ABB RAPID module: TG_Comms.sys

MODULE TG_Comms(SYSMODULE)
    !***********************************************************************
    ! TetraGen HMI request library for ABB - Phase 1 (comm core)
    !
    ! RAPID port of the FANUC KAREL request programs.
    ! Design & wire protocol: docs/abb_port_plan_v1.md
    !
    ! Loaded resident in task T_ROB1. The .tgs program modules (loaded
    ! dynamically by TG_Main in Phase 3) call the TG_* PROCs and read the
    ! shared PERS data below directly - RAPID's task-wide global scope makes
    ! every non-LOCAL symbol of a loaded module visible to all other modules.
    !
    ! Naming:  TG_*  = public API (called by TG_Main and .tgs programs)
    !          tg*   = internal helpers (LOCAL)
    !
    ! Wire protocol: byte-compatible with the FANUC TGS HMI protocol
    ! (request ids, prompts, 1-byte "0" acks, fixed-width scalars) EXCEPT
    ! frame/pose payloads, which travel as RAPID pose literals
    ! "[[x,y,z],[q1,q2,q3,q4]]" with a normalized quaternion (plan 4.5).
    !
    ! Tool/frame parameter style (plan 7.6, decided 2026-08-28): the pose-
    ! reporting request PROCs take explicit \Tool/\WObj PERS parameters
    ! (option b - the frame is visible at every call site, and a PERS
    ! parameter is itself a persistent reference, so it feeds CRobT
    ! directly). The FANUC-style modal numbers (nTG_ActTool/nTG_ActFrame)
    ! remain as a DEPRECATED fallback for calls that omit the arguments -
    ! kept deliberately as the back-pocket alternative; do not delete.
    !***********************************************************************

    ! ------------------------------------------------------------------
    ! Connection config. Edit from FlexPendant/RobotStudio, no code change.
    ! Virtual controller: keep "127.0.0.1". Real IRC5: the controller LAN IP.
    PERS string stTG_ServerIP:="127.0.0.1";
    PERS num nTG_Port:=2000;

    ! Settle time (s) applied after WaitRob and before every reported pose.
    ! VC measurements (findings doc): WaitRob \InPos alone left up to ~2 mm
    ! of residual convergence; 0.2 s reaches full settle (and matches the
    ! FANUC WAIT 0.20 before R_C). Tune from the data view without reloading
    ! code; on the real cell it also covers mechanical vibration damping.
    PERS num nTG_SettleTime:=0.2;

    ! ------------------------------------------------------------------
    ! Shared state: FANUC register-map equivalents (plan 4.3).
    PERS string stTG_ProgPass:="none";     ! SR[24] program name == project password
    PERS string stTG_SubName:="none";      ! SR[25] sub-routine token
    PERS string stTG_RobStatus:="Ok";      ! SR[23] robot status string
    PERS string stTG_ProgName:="none";     ! prog name received by TG_ReqFileTransfer
    PERS num nTG_ProgSel:=0;               ! R[188] 1=run .tgs program, 2=camera calibration
    PERS num nTG_FtpStatus:=0;             ! R[189] file transfer ok
    PERS num nTG_PassOK:=0;                ! R[200] password correct
    PERS num nTG_DryRun:=0;                ! R[199] dry-run flag
    PERS num nTG_DoCapture:=0;             ! R[197] do-capture flag; 2 = robot-side abort sentinel (matrix I4)
    PERS num nTG_CaptureOK:=0;             ! R[196] capture succeeded
    PERS num nTG_GlobalCapOK:=0;           ! R[187] global captures done status
    PERS num nTG_WeldStatus:=0;            ! R[198] 0=skip weld, 1=weld, 2=abort program
    PERS num nTG_UdwpFlag:=0;              ! R[170] user-defined weld params flag
    PERS num nTG_WelderType:=0;            ! 1=Miller, 2=FroniusTPSi (KAREL local var)
    PERS num nTG_WeldProc:=0;              ! R[171] weld procedure number
    PERS num nTG_WireFeed:=0;              ! R[172] wire feed speed
    PERS num nTG_ArcLength:=0;             ! R[173] arc length
    PERS num nTG_ArcControl:=0;            ! R[174] arc control
    PERS num nTG_TravelSpeed:=0;           ! R[175] travel speed

    ! ---- WS3/WS4 (2026-09-20): the values ABB needs and FANUC does not -----
    ! ABB takes weld parameters from the PROGRAM, not from a numbered schedule
    ! on the controller, so the HMI must serve the whole set on every weld -
    ! see the R_W_P note in TG_ReqWeldParams. Two additions carry what the
    ! FANUC wire never had to:
    !
    ! nTG_WeldSched is the POWER SOURCE's program / characteristic number,
    ! which lands in welddata main_arc.sched. It is NOT the FANUC "schedule
    ! number" of WELD START[proc,sched] (that selects a row in an ArcTool
    ! schedule file, a concept ABB has no equivalent of); it is the number the
    ! Fronius/Miller uses to pick a synergic line. MONARCH's own welddata
    ! records carry 1, 2 and 4 here.
    PERS num nTG_WeldSched:=0;             ! -> welddata main_arc.sched
    ! The seam phases: the parts of a weld either side of the steady arc.
    ! MONARCH's mDeclarations.sys carries ~15 distinct seamdata records that
    ! differ almost entirely in these, so a preset that cannot express them
    ! cannot reproduce their welds. Times in SECONDS, wire feeds in IPM and
    ! volts absolute - the same units the rest of this wire uses; TG_Weld.sys
    ! does the conversion, this module only stores.
    PERS num nTG_PurgeTime:=0;             ! -> seamdata purge_time
    PERS num nTG_PreflowTime:=0;           ! -> seamdata preflow_time
    PERS num nTG_PostflowTime:=0;          ! -> seamdata postflow_time
    PERS num nTG_BurnbackTime:=0;          ! -> seamdata bback_time
    PERS num nTG_CraterFillTime:=0;        ! -> seamdata fill_time
    PERS num nTG_CraterFillWireFeed:=0;    ! -> seamdata fill_arc.wirefeed
    PERS num nTG_CraterFillVolts:=0;       ! -> seamdata fill_arc.voltage
    PERS num nTG_IgnitionWireFeed:=0;      ! -> seamdata ign_arc.wirefeed
    PERS num nTG_IgnitionVolts:=0;         ! -> seamdata ign_arc.voltage

    ! Phase 7 (2026-09-04): pendant touch-up offset mirror (FANUC R[180..182],
    ! r_w_f.kl of the same date). The HMI pushes its stored per-weld touch-up
    ! offset on EVERY weld-frame reply - weld, skip and abort alike -
    ! so this always mirrors HMI state for the weld last served ("registers
    ! are a mirror, never a store", HMI docs/pendant_touchup_hmi_plan_v1.md).
    ! RECEIVE-AND-STORE ONLY: nothing on the ABB side consumes it yet - the
    ! FlexPendant entry/send path (FANUC R_O_T, id 20) is not ported.
    ! Units: INCHES verbatim off the wire (their D4), converted nowhere.
    PERS pos posTG_Touchup:=[0,0,0];       ! R[180..182] X/Y/Z, inches

    ! Phase 6: R_W_S weld statistics. No FANUC register equivalent - KAREL
    ! read the ArcTool record $AWEWELDSTAT[1] directly (R_W_S.kl). An IRC5
    ! has no drop-in equivalent of that record, so the .tgs program writes
    ! these three PERS just before calling TG_ReqWeldStats.
    ! TODO: DUMMY VALUES - the .tgs programs currently write fixed numbers to
    ! mimic the sensing. Producing REAL values is its own task; the candidate
    ! sources are listed in docs/abb_weld_stats_port_v1.md section 6. Only the
    ! source of the numbers changes then - the wire below is final.
    ! Units are fixed by the HMI, not by us: distance in mm (it divides by
    ! 25.4 for its analytics, which take inches) and time in seconds.
    PERS num nTG_WeldDist:=0;              ! $WELD_DIST   welded distance, mm
    PERS num nTG_ArcOnTime:=0;             ! $ARC_ON_TIME arc-on time, s
    ! 1 = the arc really ran. The HMI tests this for equality with 1, so it is
    ! a FLAG here, never a count - see the doc's 1.4 for why that distinction
    ! is not merely theoretical on the FANUC side.
    PERS num nTG_SuccArcEnd:=0;            ! $SUCC_AE

    ! Phase 5 (touch-up/retrieval doc section 4): 1 = an operator-edited
    ! .tgs module was detected at unload and staged in HOME:/TGS/edited/
    ! for the HMI's "Retrieve robot program from controller". No FANUC
    ! register equivalent (FANUC needs none: its MD: memory device serves
    ! the touched-up program directly). Set by tgSaveEditedModule
    ! (TG_Main); cleared by the HMI/tg_retrieve.py after a successful
    ! retrieval (RWS symbol write) - the robot never clears it.
    PERS num nTG_ProgEdited:=0;

    ! Frames received from the HMI (FANUC PR[5]/UFRAME[5], PR[6]/UFRAME[6]).
    ! Request PROCs write .oframe; the .tgs program references these wobjs in
    ! its move instructions - no separate "activate" step exists or is needed
    ! FOR THE TWO BASE-REFERENCED OBJECTS. The coordinated shape is another
    ! story: its station must be an ACTIVE mechanical unit (ActUnit) before
    ! a move - or a CRobT - in that work object resolves. That is one of the
    ! coordinated prerequisites still open; see the WIP block below.
    !
    ! THE RULE (weld_frame_update_strategy_v1, 2026-09-03).
    ! A request writes .oframe, ALWAYS - one write target, no case to
    ! detect here. What the HMI SENDS branches on one thing only: whether
    ! the weld is coordinated.
    !
    !   NOT COORDINATED - static table, OR indexed on a 1-/2-axis
    !   positioner that does not move during the weld:
    !       ufprog TRUE, ufmec "", uframe identity
    !       oframe <- the CAD/part frame W.R.T. THE ROBOT BASE
    !       (exactly what the HMI sends FANUC today)
    !
    !   COORDINATED MOTION - WORK IN PROGRESS, see the declaration below:
    !       ufprog FALSE, ufmec "<station>", uframe computed live by the
    !       controller from the station angles (the declared one ignored)
    !       oframe <- OPEN: the part W.R.T. THE POSITIONER FRAME, or a
    !       DISPLACEMENT in that frame, which is what the HMI's own
    !       (unfinished, untested) coordinated FANUC path computes today
    !
    ! Writing THE SERVED FRAME to uframe is never right. Coordinated: the
    ! controller ignores uframe outright (plan E28), so the write is a
    ! SILENT no-op - finding F-2's failure mode. Not coordinated: uframe is
    ! identity, so writing oframe is the same geometry anyway, because
    ! motion and CRobT both see only the product uframe*oframe.
    !
    ! BUT "uframe is identity" is a claim about the LIVE PERS VALUE, not
    ! about the declarations below. A PERS keeps whatever it was last
    ! assigned - across program loads, and across a saved station - so a
    ! controller that ever ran the pre-2026-09-03 code, which served the
    ! frame INTO uframe, still holds that frame there. Compose it with the
    ! new oframe write and every pose is double-transformed silently, while
    ! a pendant watch on oframe shows exactly the expected numbers.
    ! => AN EXPORTED PROGRAM MUST ASSIGN uframe:=IDENTITY AT ENTRY, next to
    ! its .oframe nominal, for every base-referenced work object it uses.
    ! That is a one-time normalization of an assumption, NOT a frame write,
    ! and it is the one legitimate reason to touch uframe at all.
    ! TD05Test.mod and TD05Weld.mod both do it; THE WELD PLANNER ABB
    ! EXPORTER MUST TOO.
    !
    ! ONE DECLARATION PER SHAPE - ufprog/ufmec ARE NEVER WRITTEN AT RUNTIME.
    ! The two shapes are separate symbols, so a program picks one by PASSING
    ! it (\WObj:=...) rather than by mutating a record. Reasons, in order:
    !   - runtime ufmec re-binding is unverified and unusual; declaring each
    !     shape once makes the question moot;
    !   - a program mixing indexed and coordinated welds would otherwise
    !     have to reassign mid-run, which is exactly the look-ahead hazard
    !     tracked as O-3 (a PERS write landing after RAPID has already
    !     prepared queued instructions);
    !   - robtargets bind by NAME, so a record whose kind changes mid-program
    !     makes the same named target mean different things at different
    !     points - and a pendant watch shows one mutating record;
    !   - the static shape stays byte-identical to what a VC has accepted.
    ! An exported program therefore assigns only frame COMPONENTS at entry -
    ! .uframe identity and .oframe nominal - never ufprog/ufmec.
    ! EXCEPTION (2026-09-23, VC-proven): wobjTG_WeldActStn below is bound
    ! at run time by TG_ActMechUnit - once, at module entry, before any
    ! motion - so one coordinated program can run on either station. It is a
    ! separate record, always coordinated, so none of the reasons above bite.
    ! NOTE Accepted cost: ufprog/ufmec correctness
    ! now lives on the controller, the same trust model as tTG_Weld - a
    ! wrong ufmec here is a silent wrong-station weld, so treat these as
    ! cell configuration and verify them when commissioning.
    !
    ! For an INDEXED weld the served frame describes the part AT THE ANGLE
    ! THE WELD PLANNER AUTHORED for that weld: the HMI rotates its
    ! localization result from the capture angle to the weld's
    ! tool_path_parameters positioner_angle - bTpos * Rz(dtheta) *
    ! inverse(bTpos) - and NEVER reads the robot's actual station position.
    ! So the served value does not depend on when the request runs, and the
    ! real requirement is that THE PROGRAM'S INDEX EQUALS THE ANGLE THE
    ! PLANNER AUTHORED (true by construction for an exported program).
    ! Keep the safe order regardless: index, then request the frame, then
    ! weld. And once a frame has been served, do not re-assign either
    ! component before the weld that consumes it.
    !
    ! ---- Non-coordinated: static table, or indexed on a positioner -------
    ! Base-referenced. Identity uframe, so uframe*oframe = oframe = whatever
    ! the HMI serves. These are also the standalone/VC defaults.
    PERS wobjdata wobjTG_Cam:=[FALSE,TRUE,"",[[0,0,0],[1,0,0,0]],[[0,0,0],[1,0,0,0]]];
    PERS wobjdata wobjTG_Weld:=[FALSE,TRUE,"",[[0,0,0],[1,0,0,0]],[[0,0,0],[1,0,0,0]]];

    ! ---- Coordinated motion, one work object per station -----------------
    ! WORK IN PROGRESS on both sides of the wire, 2026-09-03. These are the
    ! declared shapes only; nothing in this repo references them yet, and the
    ! prerequisites listed at the end of this block are all still open.
    ! UPDATE 2026-09-12: the oframe CONVENTION is no longer open - it is
    ! ABSOLUTE, see below - and the PC-side exporter now passes these records
    ! by name (curobo_suite D47). The prerequisites below are unchanged and
    ! still open, and nothing here has been loaded on a controller.
    !
    ! ufprog FALSE + ufmec => the controller derives uframe live from the
    ! station angles and IGNORES the declared uframe, which is why it is
    ! left identity. oframe is the component TG_ReqWeldFrame writes.
    !
    ! COMMENT THESE DECLARATIONS OUT WHEN THE TEST CELL HAS NO EXTERNAL AXIS,
    ! or change "STN1"/"STN2" to the mechanical units of the setup being
    ! tested - and comment out the second one on a single-station cell.
    ! Each name must exist in this controller's MOC configuration, and the
    ! phase 1-6 validation VC (RW6.15.08/IRB4600) has no positioner at all.
    ! THIS FILE IS THE SHARED SYSMODULE: if a controller rejects an
    ! unresolvable ufmec at load or at Check Program, it takes the ALREADY
    ! VALIDATED non-coordinated path down with it - and there are now TWO
    ! names that can do that. One "!" in front of each declaration line is
    ! the whole rollback. Note the asymmetry - an unresolvable name fails
    ! loudly, while a wrong-but-resolvable one is a silent wrong-station
    ! weld, so verify BOTH names at commissioning. Two declared stations
    ! make that silent case reachable on a correctly built cell for the
    ! first time: STN1/STN2 transposed welds the right geometry on the
    ! wrong table, where with one station declared a mix-up could only ever
    ! fail loudly.
    ! NOTE NOT YET LOADED ON A CONTROLLER. Only the static shape above has been
    ! (LOCAL PERS wobjdata accepted as a \WObj argument, RW6.15.08/IRB4600,
    ! Check Program clean). Bundle this with the coordinated VC load-check.
    !
    ! WHAT THIS oframe CARRIES - RESOLVED 2026-09-12 as ABSOLUTE: the
    ! CORRECTED PART POSE IN THE WORK OBJECT'S USER FRAME, which for these
    ! records is the station. Not a displacement. Decision is curobo_suite
    ! plan D47; full reasoning and the rejected alternative are in
    ! curobo_suite docs/abb_coordinated_hmi_frame_contract_v1.md.
    !
    ! The deciding argument is SLOT COUNT, not geometry. FANUC can afford a
    ! displacement because it has TWO runtime registers - the absolute goes
    ! to the UFRAME PR and the delta to the OFFSET PR, two slots with two
    ! meanings that cannot collide. Here there is ONE writable frame, and
    ! .oframe is ALSO where the non-coordinated absolute lands, because
    ! TG_ReqWeldFrame writes it unconditionally on whatever it is handed
    ! (the O-1 resolution). Under a displacement convention that one slot
    ! would mean "absolute" for wobjTG_Weld and "delta" for
    ! wobjTG_WeldStn<n>, with NO ERROR when the two are swapped. Absolute
    ! gives one sentence covering both records and keeps RAPID free of case
    ! detection. ABB's own MultiMove manual reads the same way: its
    ! wobj_stn1 example puts the part's mounting offset in oframe.
    !
    ! A displacement is NOT geometrically impossible - it works if the
    ! exporter re-encodes the robtargets into the positioner flange frame,
    ! which is exactly what the FANUC path does. So this was a cost and
    ! coupling decision, not a correctness one, and section 7 of
    ! docs/abb_coordinated_weld_hmi_plan_v1.md (curobo_suite) records what
    ! would reopen it: a decision to keep getWeldFrameToSendToRobot
    ! brand-blind.
    !
    ! WHAT THE HMI STILL HAS TO DO. RobotCell::getWeldFrameToSendToRobot is
    ! brand-agnostic today and returns
    ! Weld::GetCoordinatedOffsetInPositionerFrame - the FANUC DISPLACEMENT -
    ! for every coordinated weld. Fed to TG_ReqWeldFrame that produces a
    ! module which loads, runs, and welds in the wrong place with no error.
    ! That call site must branch on brand IN THE SAME CHANGE that enables
    ! coordinated ABB welds. The correct value is the existing offset
    ! composed onto the nominal: offset_in_pos * (inv(P) * C_nom) =
    ! inv(P) * C_cor, exact, and C_nom cancels.
    !
    ! Prerequisites, none of them closed (all WIP):
    !   - ActUnit for the station, and whether it is a mechanical unit in
    !     the robot's own motion task or a MultiMove group (SyncMoveOn);
    !   - real extjoint values for the station axes in every robtarget -
    !     the exporter writes 9E9 for axes it does not command (plan D5);
    !   - the controller's STN1 and STN2 BASE FRAMES must EACH agree with
    !     the positioner calibration the PC uses. A disagreement is a silent
    !     rigid offset on every coordinated weld on THAT station - E47 one
    !     level up, and a bigger risk than a mistyped ufmec. Two stations is
    !     two independent calibrations to verify, not one checked twice.
    PERS wobjdata wobjTG_WeldStn1:=[FALSE,FALSE,"STN1",[[0,0,0],[1,0,0,0]],[[0,0,0],[1,0,0,0]]];
    ! Station 2 (D4's two-station template). Same shape, different ufmec, and
    ! a SEPARATE resident symbol for exactly the reason Stn1 is separate from
    ! wobjTG_Weld: ufmec is baked into the record and is never re-bound at
    ! runtime, so one work object cannot serve both stations. Each station is
    ! declared once here and an exported program picks one BY PASSING IT -
    ! TG_ReqWeldFrame writes .oframe on whatever it is handed - so which
    ! station a weld belongs to is expressed entirely at the call site:
    !     TG_ReqWeldFrame \Tool:=tTG_Weld \WObj:=wobjTG_WeldStn2;
    ! The two oframes are independent slots and serving one never touches the
    ! other, so a program alternating stations does not disturb a frame it
    ! already holds for the other one. Everything above applies unchanged:
    ! same oframe convention (ABSOLUTE, resolved 2026-09-12), same
    ! prerequisites, same rollback.
    !
    ! TWO PREREQUISITES THAT ONLY EXIST ONCE THERE ARE TWO STATIONS, both
    ! read off the MONARC teardown of a real IRBP D600 two-station cell
    ! (customer_specific/monarc/, joint_limits.md and monarc_cell_teardown.html):
    !   - THE STATIONS CANNOT BOTH BE ACTIVE. Five positioner motors share
    !     three drives through contactors K1-K5, so ActUnit STN2 requires
    !     DeactUnit STN1 first. Declaring both work objects is fine -
    !     declaring is not activating - but only the ACTIVE station's object
    !     resolves for a move or a CRobT. A two-station program brackets
    !     each station's work in ActUnit/DeactUnit.
    !   - THE extjoint SLOTS ARE SHARED. eax_b/eax_c are ARM1/PLATE1 or
    !     ARM2/PLATE2 depending on which unit is active, because the logical
    !     axis numbers are reused. A robtarget carried from a station-1
    !     program into a station-2 one commands station 2's axes to station
    !     1's angles WITHOUT COMPLAINT. That lands on the exporter (plan
    !     D5), not here, but it is the same silent-wrong-station family as
    !     a transposed ufmec.
    ! NOTE "STN1"/"STN2" are the actual configured unit names in that cell,
    ! which is the best evidence available that these are the right strings -
    ! but neither has been checked against the target controller's MOC, so
    ! treat both as unverified until commissioning.
    ! NOTE The MONARC feasibility note proposes moving the coordinated objects
    ! out into a per-cell TG_Frames.sys adapter, on the grounds that station
    ! names are cell configuration rather than generic core. That split has
    ! not been taken; if it is, both declarations move together.
    PERS wobjdata wobjTG_WeldStn2:=[FALSE,FALSE,"STN2",[[0,0,0],[1,0,0,0]],[[0,0,0],[1,0,0,0]]];

    ! ---- Coordinated motion, "the station at the robot" -------------------
    ! 2026-09-23, VC-proven: ONE coordinated work object for
    ! whichever station is presented, so a coordinated program names no
    ! station and can run on both. Declared UNBOUND (ufmec ""): TG_ActMechUnit
    ! (TG_Cell.sys) writes ufmec from the SAME decision that activates the
    ! unit, on every call, before the program's first motion. Measured on the
    ! ProjectMonarch VC (RW 6.15, socket plan V-36):
    !   - ufmec "" loads; used unbound, CRobT stops the program (41450);
    !   - bound to the active station, a coordinated MoveL follows it: the
    !     station frame turned exactly with the chuck (9.961 deg for 9.961);
    !   - bound to the INACTIVE station, CRobT only LOGS 50066 and returns a
    !     pose that is not station-relative - execution continues - and the
    !     next coordinated move stops with 50066. No wrong-station motion;
    !   - a unit name the controller does not have stops the program (41450).
    ! The per-station records above stay for programs that name a station.
    PERS wobjdata wobjTG_WeldActStn:=[FALSE,FALSE,"",[[0,0,0],[1,0,0,0]],[[0,0,0],[1,0,0,0]]];

    ! No coordinated CAMERA work object, deliberately. Captures stay
    ! base-referenced on ABB exactly as on FANUC, so the HMI's scan and
    ! registration path is one code path across both brands (owner call,
    ! 2026-09-03). What that costs is a known, accepted accuracy item, not an
    ! oversight. See weld_frame_update_strategy_v1.md section 5, and for the
    ! two ways in if measurement later says it matters.
    !
    ! CORRECTION 2026-09-12 - the conditioning argument this note used to
    ! make does not survive measurement, and the convention it hedged on is
    ! now settled (see the coordinated block above). It read:
    !
    !   "What that costs depends on the open convention question above.
    !    Under the ABSOLUTE reading the PC's positioner model enters as a
    !    single left-multiply - inverse(plate_pc(theta_s)) * P_base - so a
    !    calibration error there lands on the weld at full magnitude. Under
    !    the DISPLACEMENT reading it enters as a conjugation that cancels at
    !    zero correction, which is the better-conditioned arithmetic."
    !
    ! Tested rather than argued. Model the station miscalibration as
    ! plate_ctrl(theta) = Y * plate_pc(theta) with Y = 3 mm + 0.2 deg, over a
    ! 7-sample 2-axis sweep with the tilt parked at 37 deg. Both conventions
    ! are wrong by EXACTLY THE SAME AMOUNT - 7.047 mm with no correction,
    ! 7.056 mm with a 2.6 mm correction - and both are exact (1e-12 mm) on a
    ! calibrated station. They are algebraically identical under that error
    ! mode, because Y left-multiplies the whole chain either way:
    ! plate_ctrl(theta) * oframe * p == plate_ctrl(theta) * delta * q for the
    ! corresponding point encodings.
    !
    ! The conjugation DOES cancel at zero correction - but what it cancels is
    ! the CORRECTION term, and the dominant term is the part's nominal
    ! placement, which crosses the PC/controller frame boundary exactly once
    ! in both conventions. So displacement buys no robustness here, and the
    ! absolute convention costs none.
    !
    ! WHAT THIS DOES NOT COVER, and is still open: an error in how the PC
    ! models the plate's MOTION - axis direction or offset, i.e. a
    ! theta-DEPENDENT mismatch rather than a constant Y. That was not tested
    ! and is a different question. If that is the real concern, measure it
    ! the same way before acting on it; the constant-Y result says nothing
    ! about it either way.

    ! Tools (FANUC UT[2] camera / UT[8] torch).
    ! TODO: DUMMY VALUES - replace with the calibrated tooldata of the real cell.
    PERS tooldata tTG_Cam:=[TRUE,[[0,0,100],[1,0,0,0]],[1,[0,0,50],[1,0,0,0],0,0,0]];
    PERS tooldata tTG_Weld:=[TRUE,[[0,0,200],[1,0,0,0]],[1,[0,0,100],[1,0,0,0],0,0,0]];

    ! DEPRECATED (plan 7.6, decided 2026-08-28) - FANUC modal
    ! UTOOL_NUM/UFRAME_NUM emulation: the .tgs program selects the active
    ! tool/frame BY NUMBER; tgSendPose resolves the number to the LIVE
    ! tooldata/wobjdata at read time. Superseded by explicit \Tool/\WObj
    ! PERS parameters on the request PROCs (style b), which make the frame
    ! visible at the call site instead of hidden global state. Only used
    ! when a request is called WITHOUT the arguments. Kept deliberately as
    ! the back-pocket alternative; do not delete.
    ! (A PERS-to-PERS copy would go stale when a request updates the frame -
    ! the same hazard FANUC handles by re-emitting UFRAME[n]=PR[n] after
    ! every frame-PR-writing routine. Numbers need no refresh.)
    PERS num nTG_ActTool:=8;               ! UTOOL_NUM:  2=camera, 8=torch
    PERS num nTG_ActFrame:=0;              ! UFRAME_NUM: 5=camera, 6=weld, else base

    ! Scratch persistents for CRobT: its \Tool/\WObj are PERS parameters
    ! (a VAR or FUNC result is rejected with Argument error 123). Only the
    ! DEPRECATED modal fallback needs them (tgActTool/tgActWobj are FUNCs,
    ! their results are values); the explicit style passes the caller's
    ! PERS parameters straight to CRobT, no scratch copy involved.
    ! tgSendPose refreshes them from the live data on every fallback call,
    ! so they cannot go stale. Internal - never reference in .tgs programs.
    LOCAL PERS tooldata tTG_Scratch:=[TRUE,[[0,0,200],[1,0,0,0]],[1,[0,0,100],[1,0,0,0],0,0,0]];
    LOCAL PERS wobjdata wobjTG_Scratch:=[FALSE,TRUE,"",[[0,0,0],[1,0,0,0]],[[0,0,0],[1,0,0,0]]];

    ! ------------------------------------------------------------------
    ! Socket state. Lifecycle owned by TG_Main via TG_SocketCom/TG_SocketDisc;
    ! .tgs programs must never touch these directly.
    LOCAL VAR socketdev tg_server_socket;
    LOCAL VAR socketdev tg_client_socket;
    LOCAL VAR string tg_client_ip:="";


    !===================================================================
    ! Socket lifecycle (FANUC: SOCKET_COM / SOCKET_DISC)
    !===================================================================

    PROC TG_SocketCom()
        ! FANUC: SOCKET_COM - (re)start the server and wait for the HMI client.
        ! SocketClose is safe on sockets that were never opened (RoboDK driver
        ! uses the same close-before-create pattern on RW5/6).
        SocketClose tg_server_socket;
        SocketClose tg_client_socket;
        SocketCreate tg_server_socket;
        SocketBind tg_server_socket,stTG_ServerIP,nTG_Port;
        SocketListen tg_server_socket;
        TPWrite "TG: waiting for HMI on port "\Num:=nTG_Port;
        SocketAccept tg_server_socket,tg_client_socket\ClientAddress:=tg_client_ip,\Time:=WAIT_MAX;
        TPWrite "TG: HMI connected: "+tg_client_ip;
    ERROR
        ! Error matrix F-A/I1: RAPID's retry counter is bounded by the
        ! system parameter "No Of Retry" (default 4) - without
        ! ResetRetryCount a handful of consecutive failures would stop the
        ! whole server loop. Resetting makes this reconnect loop indefinite
        ! (same idiom as the RoboDK driver). Pacing comes from WaitTime /
        ! the blocking SocketAccept, so this cannot busy-loop.
        IF ERRNO=ERR_SOCK_TIMEOUT THEN
            ResetRetryCount;
            RETRY;
        ELSEIF ERRNO=ERR_SOCK_CLOSED THEN
            SocketClose tg_server_socket;
            SocketClose tg_client_socket;
            WaitTime 2;
            ResetRetryCount;
            RETRY;
        ENDIF
    ENDPROC

    PROC TG_SocketDisc()
        ! FANUC: SOCKET_DISC - drop the HMI connection (and the listener; it is
        ! re-created by the next TG_SocketCom). WaitTime lets the TCP stack
        ! release the port before rebinding (RoboDK COM_End pattern).
        SocketClose tg_server_socket;
        SocketClose tg_client_socket;
        WaitTime 2;
        TPWrite "TG: socket disconnected";
    ENDPROC


    !===================================================================
    ! Wire-protocol helpers (plan 4.4)
    !===================================================================

    LOCAL PROC tgCycleAbort()
        ! FIX 2026-08-28 (error-recovery matrix F-F): bottom-level recovery
        ! for wire errors. VC evidence (kill test, RW 6.15): an unhandled
        ! error does NOT propagate through the late-binding call
        ! (%stTG_ProgName%) - the program STOPPED at the failing
        ! SocketReceive (events 41595/40228), so the tgRunTgsProgram /
        ! tgMainCycle handlers can never see a wire error raised inside a
        ! .tgs run. Recover where the error is born instead: log, drop the
        ! sockets, ExitCycle. PP moves to the start of main, which begins
        ! with TG_SocketDisc and loops back to accept - no propagation
        ! involved, works from any call depth (VC-validated 2026-08-28).
        ! VC-observed: ExitCycle's PP move does NOT drop \Dynamic modules
        ! (unlike a FlexPendant/RobotStudio PP-to-main) - the leftover is
        ! handled next cycle by the ERR_LOADED reload path (matrix I2),
        ! also VC-validated in exactly this scenario.
        ! Called ONLY from the wire helpers' ERROR handlers below.
        ! To stop instead of recovering, replace ExitCycle below with:
        !   EXIT             - terminates execution (FANUC abort)
        !   Stop             - halts, resumable with Start (FANUC pause)
        !   Stop; ExitCycle; - halt for the operator, clean restart on Start
        TPWrite "TG: cycle error, ERRNO = "\Num:=ERRNO;
        TPWrite "TG: wire lost - restarting cycle";
        SocketClose tg_server_socket;
        SocketClose tg_client_socket;
        ExitCycle;
    ENDPROC

    LOCAL PROC tgSendAck(string data)
        ! Robot->HMI message: send, then wait for the HMI 1-byte ack ("0").
        ! KAREL: WRITE comm_file(data) ; READ comm_file(cmd::1)
        VAR string ack;
        SocketSend tg_client_socket,\Str:=data;
        SocketReceive tg_client_socket,\Str:=ack,\Time:=WAIT_MAX;
    ERROR
        ! FIX 2026-08-28 (F-F): catch-all - any error on the wire aborts
        ! the cycle from here (see tgCycleAbort; propagation upward cannot
        ! be relied on inside a late-bound .tgs run).
        tgCycleAbort;
    ENDPROC

    LOCAL FUNC string tgPromptRecv(string prompt)
        ! HMI->robot value: send the sync prompt, then receive the payload.
        ! KAREL: WRITE comm_file(prompt) ; READ comm_file(cmd::N)
        VAR string reply;
        SocketSend tg_client_socket,\Str:=prompt;
        SocketReceive tg_client_socket,\Str:=reply,\Time:=WAIT_MAX;
        RETURN reply;
    ERROR
        ! FIX 2026-08-28 (F-F): catch-all - see tgSendAck.
        tgCycleAbort;
    ENDFUNC

    LOCAL FUNC string tgFmtReal(num v)
        ! FANUC fixed-width real: sign + 8 chars, 3 decimals, zero-padded.
        ! e.g. 905.216 -> "+0905.216", -12.5 -> "-0012.500"
        VAR string s;
        VAR num av;
        VAR num dotpos;
        av:=Abs(v);
        ! FANUC HMI rejects values >= 10000 anyway (frame limit check)
        IF av>9999.999 av:=9999.999;
        s:=NumToStr(av,3);
        ! ensure exactly 3 decimals (NumToStr may drop trailing zeros)
        dotpos:=StrFind(s,1,".");
        IF dotpos>StrLen(s) THEN
            s:=s+".000";
            dotpos:=StrFind(s,1,".");
        ENDIF
        WHILE StrLen(s)-dotpos<3 DO
            s:=s+"0";
        ENDWHILE
        ! zero-pad the integer part to a total of 8 chars
        WHILE StrLen(s)<8 DO
            s:="0"+s;
        ENDWHILE
        IF v<0 THEN
            RETURN "-"+s;
        ENDIF
        RETURN "+"+s;
    ENDFUNC

    LOCAL FUNC num tgParseReal(string s)
        ! Tolerant scalar parse; returns 0 on garbage (and reports it).
        ! Strips the FANUC-format leading "+" ("+0017.500"): an explicit plus
        ! sign is not part of a RAPID num literal, so StrToVal may reject it.
        ! (Nested IFs: RAPID AND does not short-circuit; local copy: IN
        ! parameters are not writable.)
        VAR string s2;
        VAR num v:=0;
        VAR bool ok;
        s2:=s;
        IF StrLen(s2)>0 THEN
            IF StrPart(s2,1,1)="+" THEN
                s2:=StrPart(s2,2,StrLen(s2)-1);
            ENDIF
        ENDIF
        ok:=StrToVal(s2,v);
        IF NOT ok THEN
            TPWrite "TG ERROR: bad number payload:";
            TPWrite s2;
            v:=0;
        ENDIF
        RETURN v;
    ENDFUNC

    LOCAL FUNC string tgPoseToStr(pose p)
        ! RAPID pose literal, guaranteed <= 80 chars for |trans| < 10000 mm
        ! (plan 4.5): translations 2 decimals, quaternions 6 decimals.
        VAR string s;
        s:="[["+NumToStr(p.trans.x,2)+","+NumToStr(p.trans.y,2)+","+NumToStr(p.trans.z,2)+"],[";
        s:=s+NumToStr(p.rot.q1,6)+","+NumToStr(p.rot.q2,6)+",";
        s:=s+NumToStr(p.rot.q3,6)+","+NumToStr(p.rot.q4,6)+"]]";
        RETURN s;
    ENDFUNC

    LOCAL FUNC bool tgTryStrToPose(string s,INOUT pose p)
        ! Parse "[[x,y,z],[q1,q2,q3,q4]]" into a pose; re-normalize the
        ! quaternion defensively (non-normalized orients raise error 50076
        ! when used in motion). Leaves p untouched on parse failure.
        VAR pose ptmp;
        VAR bool ok;
        ok:=StrToVal(s,ptmp);
        IF ok THEN
            ptmp.rot:=NOrient(ptmp.rot);
            p:=ptmp;
        ELSE
            TPWrite "TG ERROR: bad pose payload:";
            TPWrite s;
        ENDIF
        RETURN ok;
    ENDFUNC

    LOCAL FUNC tooldata tgActTool()
        ! DEPRECATED (plan 7.6) - modal fallback only, see nTG_ActTool.
        ! Resolve the FANUC-style active tool number to live tooldata.
        IF nTG_ActTool=2 THEN
            RETURN tTG_Cam;
        ENDIF
        RETURN tTG_Weld;
    ENDFUNC

    LOCAL FUNC wobjdata tgActWobj()
        ! DEPRECATED (plan 7.6) - modal fallback only, see nTG_ActFrame.
        ! Resolve the FANUC-style active frame number to live wobjdata.
        IF nTG_ActFrame=5 THEN
            RETURN wobjTG_Cam;
        ELSEIF nTG_ActFrame=6 THEN
            RETURN wobjTG_Weld;
        ENDIF
        RETURN wobj0;
    ENDFUNC

    LOCAL PROC tgSendPose(\PERS tooldata Tool,\PERS wobjdata WObj)
        ! Robot->HMI: current pose of the given tool in the given frame,
        ! sent as a pose literal (plan 4.5). KAREL sent Euler x,y,z,w,p,r;
        ! the Euler<->quaternion conversion now lives on the PC side.
        ! \Tool/\WObj (pass BOTH): PERS parameters are persistent
        ! references - handed to CRobT directly, so a frame updated by a
        ! request is used by the very next pose report (FANUC
        ! UFRAME[n]=PR[n] semantics included, plan 7.6 style b).
        ! Omitted -> DEPRECATED modal fallback via nTG_ActTool/nTG_ActFrame.
        VAR robtarget rt;
        VAR pose p;
        ! Never report a pose while the servos are still converging: on the
        ! VC, CRobT read right after a fine point was 1-3 mm / ~0.08 deg off
        ! the settled position (rapid_validation_findings_v1.md, 'related
        ! observation'). Captures register against this reported pose, so
        ! the error would flow into registration.
        ! Measured escalation (2026-08-28): \InPos alone shrank the error
        ! 1.3 mm -> 0.28 mm but left ~2 mm right after a move, so all three
        ! stages are applied: stop point reached, true standstill, then a
        ! settle time for residual servo creep / mechanical vibration
        ! (FANUC used WAIT 0.20 + DELAY in the same places).
        WaitRob \InPos;
        WaitRob \ZeroSpeed;
        IF nTG_SettleTime>0 WaitTime nTG_SettleTime;
        IF Present(Tool) AND Present(WObj) THEN
            rt:=CRobT(\Tool:=Tool \WObj:=WObj);
        ELSE
            ! DEPRECATED modal path (plan 7.6) - resolve the FANUC-style
            ! numbers; FUNC results are values, hence the scratch copies.
            IF Present(Tool) XOR Present(WObj) THEN
                TPWrite "TG WARNING: tgSendPose needs BOTH Tool and WObj - using modal numbers";
            ENDIF
            tTG_Scratch:=tgActTool();
            wobjTG_Scratch:=tgActWobj();
            rt:=CRobT(\Tool:=tTG_Scratch \WObj:=wobjTG_Scratch);
        ENDIF
        p.trans:=rt.trans;
        p.rot:=rt.rot;
        tgSendAck tgPoseToStr(p);
    ENDPROC


    LOCAL FUNC dnum tgHomeFreeBytes()
        ! Free bytes on HOME:, or -1 if it cannot be measured.
        ! \Mbyte then scaled in dnum: a num holds exact integers only to
        ! 8388608 (RAPID ref 3.49), far below any real byte count.
        CONST dnum BYTES_PER_MB:=1048576;
        RETURN NumToDnum(FSSize("HOME:"\Free\Mbyte))*BYTES_PER_MB;
    ERROR
        ! ERR_FILESIZE and ERR_FILEACC are recoverable (VC-proven), and
        ! losing the disk figure must not fail the cycle: ProgMemFree still
        ! answers, and it is the tighter constraint anyway.
        TPWrite "TG WARN: HOME: free space unreadable, ERRNO ="\Num:=ERRNO;
        RETURN -1;
    ENDFUNC

    LOCAL FUNC string tgFreeMemStr()
        ! The R_F_T free-space answer, in BYTES, as plain digits. The HMI
        ! parses it with std::stoull and aborts the weld session below 40000
        ! bytes (config.json,
        ! HMI_MINIMUM_STORAGE_IN_TPP_CONTROLLER_MEMORY_IN_BYTES).
        !
        ! FANUC sent VOL_SPACE of tpp:. That single FANUC resource is TWO on
        ! ABB - the disk the module is PUT to (HOME:) and the program memory
        ! TG_Main then Loads it into - so report whichever is smaller.
        ! ProgMemFree is normally the binding one by a wide margin (VC: 35 MB
        ! against 1.9 GB of HOME:), and it is what Load consumes, so a low
        ! value here is precisely the ERR_PRGMEMFULL that the HMI's check
        ! exists to pre-empt.
        !
        ! VC-proven 2026-09-04 with abb/rapid/TGFsProbe.mod:
        !   - FSSize REQUIRES \Total or \Free. A bare call raises 40764, an
        !     UNRECOVERABLE argument error no ERROR handler can catch. The
        !     manual's syntax (2.71) prints both switches as optional and is
        !     simply wrong.
        !   - the ERR_FILESIZE ceiling (8388608, the num exact-integer max)
        !     is applied AFTER the \Kbyte/\Mbyte division, and IS
        !     recoverable (ERRNO 1121). \Mbyte therefore has 8 TB of
        !     headroom; asking for bytes raises on any file system with more
        !     than 8 MB free.
        !   - FSSize does not need the path to exist, only the device prefix
        !     resolves - so plain "HOME:" cannot fail on a missing file the
        !     way HOME:/TGS/<prog>.mod could.
        VAR dnum dnFree;
        VAR dnum dnDisk;
        CONST dnum MAX_REPORT:=999999999;
        dnFree:=NumToDnum(ProgMemFree());
        dnDisk:=tgHomeFreeBytes();
        IF dnDisk>=0 AND dnDisk<dnFree dnFree:=dnDisk;
        ! Clamp before formatting. The HMI only compares this against 40000
        ! and logs it as KB, so the true magnitude buys it nothing - while a
        ! bad string is silent and fatal: std::stoull reads "3.5185E+7" as 3,
        ! and std::stoull("-1") does not fail, it returns 1.8e19. Capping at
        ! 9 digits keeps DnumToStr inside the range actually measured on the
        ! VC (plain digits at 3.5e7 and at 1.9e9) rather than trusting it at
        ! magnitudes nobody has tested.
        IF dnFree>MAX_REPORT dnFree:=MAX_REPORT;
        IF dnFree<0 dnFree:=0;
        RETURN DnumToStr(dnFree,0);
    ENDFUNC


    !===================================================================
    ! Request PROCs (priority set, plan section 1.4)
    !===================================================================

    PROC TG_ReqProgSel()
        ! FANUC: REQ_PROG_SEL - receive the mode/program selection from the
        ! HMI right after it connects. -> nTG_ProgSel (R[188])
        VAR string reply;
        VAR bool ok;
        reply:=tgPromptRecv("Give me the program ID");
        ok:=StrToVal(reply,nTG_ProgSel);
        IF NOT ok THEN
            nTG_ProgSel:=0;
            TPWrite "TG ERROR: bad program ID:";
            TPWrite reply;
        ENDIF
        TPWrite "TG: program ID = "\Num:=nTG_ProgSel;
    ENDPROC

    PROC TG_ReqEnd(\PERS tooldata Tool,\PERS wobjdata WObj)
        ! FANUC: R_E (HMI request id 100) - program end notification.
        ! Sequence: id -> current pose -> sub-routine token.
        ! \Tool/\WObj: report tool/frame for the pose (plan 7.6 style b);
        ! omitted -> DEPRECATED modal fallback. The HMI ignores every R_E
        ! pose (plan 1.4.1), so any defensible frame is acceptable here.
        ! stTG_SubName must never be empty: an empty SocketSend transmits
        ! zero bytes and the HMI recv would block forever (default "none").
        tgSendAck "100";
        tgSendPose \Tool?Tool \WObj?WObj;
        tgSendAck stTG_SubName;
        TPWrite "TG: end request served";
    ENDPROC

    PROC TG_ReqFileTransfer()
        ! FANUC: R_F_T (HMI request id 10) - the HMI transfers the .tgs
        ! program module now, then reports the transfer status and the
        ! program name. -> nTG_FtpStatus (R[189]), stTG_ProgName (SR[24];
        ! on FANUC the program name doubles as the project password).
        VAR string reply;
        tgSendAck "10";
        ! Free space on the program storage. FANUC sent VOL_SPACE of tpp:;
        ! on ABB that is min(program memory, HOME: disk) - see
        ! tgFreeMemStr, which also owns the formatting rules.
        ! In case it needs to be skipped, instead use: tgSendAck "99999999";
        tgSendAck tgFreeMemStr();
        reply:=tgPromptRecv("Give me FTP status");
        nTG_FtpStatus:=tgParseReal(reply);
        reply:=tgPromptRecv("Give me prog name");
        stTG_ProgName:=reply;
        TPWrite "TG: ftp status = "\Num:=nTG_FtpStatus;
        TPWrite "TG: prog name = "+stTG_ProgName;
    ENDPROC

    PROC TG_ReqPassCheck(\PERS tooldata Tool,\PERS wobjdata WObj)
        ! FANUC: R_P_C (HMI request id 5) - password / dry-run check.
        ! Sequence: id -> pose -> sub token -> password -> recv 2 chars
        ! (char 1 = password correct, char 2 = dry run).
        ! \Tool/\WObj: report tool/frame for the pose (plan 7.6 style b);
        ! omitted -> DEPRECATED modal fallback.
        ! -> nTG_PassOK (R[200]), nTG_DryRun (R[199])
        VAR string reply;
        tgSendAck "5";
        tgSendPose \Tool?Tool \WObj?WObj;
        tgSendAck stTG_SubName;
        tgSendAck stTG_ProgPass;
        reply:=tgPromptRecv("Give me the status");
        IF StrLen(reply)>=2 THEN
            nTG_PassOK:=tgParseReal(StrPart(reply,1,1));
            nTG_DryRun:=tgParseReal(StrPart(reply,2,1));
        ELSE
            nTG_PassOK:=0;
            nTG_DryRun:=0;
            TPWrite "TG ERROR: bad pass-check payload:";
            TPWrite reply;
        ENDIF
        TPWrite "TG: pass ok = "\Num:=nTG_PassOK;
        TPWrite "TG: dry run = "\Num:=nTG_DryRun;
    ENDPROC

    PROC TG_ReqCamFrame(\PERS tooldata Tool,\PERS wobjdata WObj)
        ! FANUC: R_C_F (HMI request id 1) - request camera frame.
        ! Sequence: id -> pose -> sub token -> recv frame (ONE pose literal,
        ! plan 4.5; KAREL received 6 prompted reals) -> recv capture flag.
        ! \Tool/\WObj (plan 7.6 style b): WObj is BOTH the report frame for
        ! the outgoing pose (which goes out in the frame's PREVIOUS value -
        ! FANUC parity, plan 1.4.1) AND the wobj whose .oframe receives the
        ! served frame, written through the PERS reference. Omitted ->
        ! DEPRECATED modal fallback; the frame lands in wobjTG_Cam.
        ! -> WObj.oframe (PR[5]/UFRAME[5]), nTG_DoCapture (R[197]; forced
        ! to 2 = abort sentinel on a bad frame payload, matrix I4)
        !
        ! The camera work object is ALWAYS the base-referenced wobjTG_Cam,
        ! for a coordinated weld as much as an indexed one - captures are
        ! taken at a standstill at one index, and keeping them
        ! base-referenced keeps the HMI's scan/registration path identical
        ! to FANUC's. There is no coordinated camera work object; see the
        ! declaration block for the accuracy item that buys.
        VAR string reply;
        VAR pose pFrame;
        VAR bool frame_ok;
        tgSendAck "1";
        tgSendPose \Tool?Tool \WObj?WObj;
        tgSendAck stTG_SubName;
        reply:=tgPromptRecv("Give me the frame");
        frame_ok:=tgTryStrToPose(reply,pFrame);
        IF frame_ok THEN
            IF Present(WObj) THEN
                WObj.oframe:=pFrame;
            ELSE
                wobjTG_Cam.oframe:=pFrame;
            ENDIF
        ENDIF
        ! The capture-status exchange must ALWAYS complete: the HMI's R_C_F
        ! handler serves the full sequence and would desync if cut short.
        reply:=tgPromptRecv("Give me capture status");
        nTG_DoCapture:=tgParseReal(reply);
        IF NOT frame_ok THEN
            ! Error matrix F-C/I4 (revised 2026-08-28: ABORT, not skip -
            ! same policy as the weld case): never proceed against a stale
            ! frame. 2 is a robot-side sentinel the HMI never sends (the
            ! wire carries only 0/1); the .tgs program checks it and aborts
            ! to R_E (FANUC LBL[101] parity).
            nTG_DoCapture:=2;
            TPWrite "TG ERROR: bad cam frame payload - aborting program";
        ENDIF
        TPWrite "TG: cam frame set, do capture = "\Num:=nTG_DoCapture;
    ENDPROC

    PROC TG_ReqCapture(\PERS tooldata Tool,\PERS wobjdata WObj)
        ! FANUC: R_C (HMI request id 2) - request camera capture at the
        ! current position. This is the ONE pose the HMI consumes (plan
        ! 1.4.1) - registration depends on Tool/WObj being the camera tool
        ! and the served camera frame.
        ! \Tool/\WObj: report tool/frame (plan 7.6 style b); omitted ->
        ! DEPRECATED modal fallback. -> nTG_CaptureOK (R[196])
        VAR string reply;
        ! FANUC: DELAY 5 (ms) "to wait for vibrations to dampen. Adjust as
        ! needed." Increase for the real cell if captures come out blurred.
        WaitTime 0.005;
        tgSendAck "2";
        tgSendPose \Tool?Tool \WObj?WObj;
        tgSendAck stTG_SubName;
        reply:=tgPromptRecv("Give me capture status");
        nTG_CaptureOK:=tgParseReal(reply);
        TPWrite "TG: capture ok = "\Num:=nTG_CaptureOK;
    ENDPROC

    PROC TG_ReqGlobalCapDone()
        ! FANUC: R_G_C_D (HMI request id 11) - all global captures done;
        ! the HMI runs global localization. -> nTG_GlobalCapOK (R[187])
        VAR string reply;
        tgSendAck "11";
        reply:=tgPromptRecv("Give me global loc status");
        nTG_GlobalCapOK:=tgParseReal(reply);
        TPWrite "TG: global loc ok = "\Num:=nTG_GlobalCapOK;
    ENDPROC

    PROC TG_ReqWeldFrame(\PERS tooldata Tool,\PERS wobjdata WObj)
        ! FANUC: R_W_F (HMI request id 4) - request weld frame.
        ! Sequence: id -> pose -> sub token -> recv frame (ONE pose literal)
        ! -> recv weld status (0=skip, 1=weld, 2=abort program)
        ! -> recv touch-up offset x/y/z (3 x 9-char reals, INCHES) into
        !    posTG_Touchup (Phase 7, 2026-09-04: receive-and-store only).
        ! \Tool/\WObj (plan 7.6 style b): WObj is BOTH the report frame for
        ! the outgoing pose AND the wobj whose .oframe receives the served
        ! frame, written through the PERS reference. Omitted -> DEPRECATED
        ! modal fallback; the frame lands in wobjTG_Weld.
        ! -> WObj.oframe (PR[6]/UFRAME[6]), nTG_WeldStatus (R[198])
        !
        ! .oframe in EVERY case, coordinated or not (see THE RULE at the
        ! top of this file), so this PROC never has to know which case it
        ! is in - and cannot, by construction: it writes .oframe on
        ! WHATEVER IT WAS HANDED, and the call site chooses.
        !     TG_ReqWeldFrame \Tool:=tTG_Weld \WObj:=wobjTG_Weld;      ! indexed
        !     TG_ReqWeldFrame \Tool:=tTG_Weld \WObj:=wobjTG_WeldStn1;  ! coord, stn 1
        !     TG_ReqWeldFrame \Tool:=tTG_Weld \WObj:=wobjTG_WeldStn2;  ! coord, stn 2
        ! What the served pose is RELATIVE TO does differ - the robot base
        ! for a non-coordinated weld (FANUC parity), the positioner frame
        ! for a coordinated one - but that follows from which work object
        ! the exporter passed, and the HMI holds the project and knows the
        ! weld's positioner group. Not this routine's business.
        ! NOTE The DEPRECATED modal fallback below writes wobjTG_Weld BY NAME,
        ! so it can only ever express the non-coordinated case. That is
        ! fine - it is the static back-pocket path - but do not extend it.
        VAR string reply;
        VAR pose pFrame;
        VAR bool frame_ok;
        tgSendAck "4";
        tgSendPose \Tool?Tool \WObj?WObj;
        tgSendAck stTG_SubName;
        reply:=tgPromptRecv("Give me the frame");
        frame_ok:=tgTryStrToPose(reply,pFrame);
        IF frame_ok THEN
            IF Present(WObj) THEN
                WObj.oframe:=pFrame;
            ELSE
                wobjTG_Weld.oframe:=pFrame;
            ENDIF
        ENDIF
        ! The weld-status and touch-up exchanges must ALWAYS complete: the
        ! HMI's R_W_F handler serves the full sequence and would desync if
        ! cut short - the abort path included.
        reply:=tgPromptRecv("Give me weld status");
        nTG_WeldStatus:=tgParseReal(reply);
        ! Phase 7: the HMI's stored touch-up offset for the weld just served
        ! (INCHES, FANUC R[180..182] parity). Stored only - nothing consumes
        ! posTG_Touchup until the FlexPendant entry path (R_O_T) is ported.
        reply:=tgPromptRecv("Give me touchup x");
        posTG_Touchup.x:=tgParseReal(reply);
        reply:=tgPromptRecv("Give me touchup y");
        posTG_Touchup.y:=tgParseReal(reply);
        reply:=tgPromptRecv("Give me touchup z");
        posTG_Touchup.z:=tgParseReal(reply);
        IF NOT frame_ok THEN
            ! Error matrix F-C/I4: never weld against a stale frame. A
            ! malformed frame payload forces the abort path (decision:
            ! abort program, not skip weld - safer for welding). The .tgs
            ! program sees nTG_WeldStatus=2 -> R_E, FANUC LBL[101] parity.
            nTG_WeldStatus:=2;
            TPWrite "TG ERROR: bad weld frame payload - aborting program";
        ENDIF
        TPWrite "TG: weld frame set, weld status = "\Num:=nTG_WeldStatus;
        TPWrite "TG: touchup offset (in) = "\Pos:=posTG_Touchup;
    ENDPROC

    PROC TG_ReqWeldParams()
        ! FANUC: R_W_P (HMI request id 14) - welding parameters.
        !
        ! WARNING: **The ABB wire is NOT the FANUC one, and deliberately so
        ! (WS3/WS4, 2026-09-20).** On FANUC the values live in an ArcTool
        ! schedule file on the controller and the program points at it with
        ! WELD START[proc,sched]; the HMI only had to send anything at all
        ! when the operator ticked "user-defined weld parameters", which is
        ! why everything below the travel speed used to sit behind
        ! IF nTG_UdwpFlag=1.
        !
        ! ABB has no such file. welddata/seamdata are ordinary RAPID data
        ! passed to the arc instructions, so whatever the HMI does not send,
        ! nothing supplies. Keeping the FANUC shape produced the defect this
        ! change fixes: a weld bound to a PRESET (UDWP=0) got travel speed
        ! and nothing else, TG_ApplyWeldParams fell back to the placeholder
        ! wdTG_Lib entry, and the weld ran at weld_speed 0.
        !
        ! So every value is now served on EVERY weld, and nTG_UdwpFlag stops
        ! being a branch: it is provenance only, telling the pendant log (and
        ! anyone reading it) whether these numbers came from the operator's
        ! overrides or from the weld's preset. The HMI decides which source
        ! to read; the robot just applies what arrives.
        !
        ! Sequence (each line is one prompt/reply round trip):
        !   UDWP flag, travel speed, welder type, proc, wire feed,
        !   arc length, arc control, weld schedule, seam phases
        !
        ! The seam phases arrive as ONE bracketed message rather than nine
        ! round trips - the same batching the frame requests already use
        ! ("Give me the frame" replaced KAREL's six x..r exchanges).
        VAR string reply;
        VAR num seam{9};
        VAR bool seam_ok;
        tgSendAck "14";
        reply:=tgPromptRecv("Give me UDWP flag");
        nTG_UdwpFlag:=tgParseReal(reply);
        reply:=tgPromptRecv("Give me travel speed");
        nTG_TravelSpeed:=tgParseReal(reply);
        reply:=tgPromptRecv("Give me welder type");
        nTG_WelderType:=tgParseReal(reply);
        reply:=tgPromptRecv("Give me proc");
        nTG_WeldProc:=tgParseReal(reply);
        reply:=tgPromptRecv("Give me wire feed speed");
        nTG_WireFeed:=tgParseReal(reply);
        reply:=tgPromptRecv("Give me arc length");
        nTG_ArcLength:=tgParseReal(reply);
        reply:=tgPromptRecv("Give me arc control");
        nTG_ArcControl:=tgParseReal(reply);
        reply:=tgPromptRecv("Give me weld schedule");
        nTG_WeldSched:=tgParseReal(reply);
        reply:=tgPromptRecv("Give me seam phases");
        seam_ok:=StrToVal(reply,seam);
        IF seam_ok THEN
            nTG_PurgeTime:=seam{1};
            nTG_PreflowTime:=seam{2};
            nTG_PostflowTime:=seam{3};
            nTG_BurnbackTime:=seam{4};
            nTG_CraterFillTime:=seam{5};
            nTG_CraterFillWireFeed:=seam{6};
            nTG_CraterFillVolts:=seam{7};
            nTG_IgnitionWireFeed:=seam{8};
            nTG_IgnitionVolts:=seam{9};
        ELSE
            ! Zero the whole block rather than leave the PREVIOUS weld's
            ! phases standing: these are PERS, so a half-parsed payload that
            ! left them alone would silently weld this seam with the last
            ! one's crater fill. Zero is also what "no seam phases" means
            ! everywhere else on this path, so TG_ApplyWeldParams needs no
            ! special case. A malformed payload is a wire defect, not an
            ! operator choice, so it is loud.
            nTG_PurgeTime:=0;
            nTG_PreflowTime:=0;
            nTG_PostflowTime:=0;
            nTG_BurnbackTime:=0;
            nTG_CraterFillTime:=0;
            nTG_CraterFillWireFeed:=0;
            nTG_CraterFillVolts:=0;
            nTG_IgnitionWireFeed:=0;
            nTG_IgnitionVolts:=0;
            TPWrite "TG ERROR: bad seam phase payload, phases zeroed:";
            TPWrite reply;
        ENDIF
        TPWrite "TG: weld params, UDWP = "\Num:=nTG_UdwpFlag;
    ENDPROC

    PROC TG_ReqWeldStats()
        ! FANUC: R_W_S (HMI request id 13) - welding stats, called once per
        ! weld right after WELD END (sample TD05tRJYQd.ls lines 223 / 392).
        ! Sequence: id -> "dist,arc_on_time,succ_ae" as ONE message. No pose,
        ! no sub token - the simplest request in the family.
        !
        ! The three values are read from the PERS above (set by the .tgs
        ! program just before the call), mirroring KAREL's three GET_VARs of
        ! $AWEWELDSTAT[1].
        !
        ! Number format: tgFmtReal ("+0200.000") - the signed zero-padded
        ! field every other scalar on this wire already uses. KAREL used
        ! CNV_REAL_STR(v,8,3), which blank-pads to a MINIMUM width with at
        ! least one leading blank (" 200.000") and emits no "+". Deliberate
        ! deviation, safe in both consumers: the HMI parses this CSV with
        ! std::stringstream >> double (FANUCRobot::ReceiveWeldingStats),
        ! which skips leading whitespace and accepts a leading "+", and so
        ! does Python float(). Keeping one real format across the port is
        ! worth more than byte parity on a field nobody compares bytewise.
        !
        ! What the HMI does with it (RobotCell.cpp case RequestWeldingStats):
        ! converts dist mm -> inches (/25.4) and, ONLY IF succ_ae equals 1,
        ! inserts a weld-analytics row (length_in, arc_on_sec). succ_ae = 0
        ! is received and discarded - that is the dry-run / no-arc path.
        VAR string stats;
        stats:=tgFmtReal(nTG_WeldDist)+","+tgFmtReal(nTG_ArcOnTime)+","+tgFmtReal(nTG_SuccArcEnd);
        tgSendAck "13";
        tgSendAck stats;
        TPWrite "TG: weld stats "+stats;
    ENDPROC

ENDMODULE
